{attribute 'GeneratedUsingTerminal: EL2002--0000'}
{attribute addProperty BoxType "EL2002--0000"}
{attribute addProperty Id "WcStateAT %I*BOOL1"}
{attribute addProperty CRC "187373305"}
{attribute addProperty Size "1"}
TYPE WcState_0B2B16F9 :
STRUCT
	{attribute addProperty Name "WcState"}
	WcState AT %I* : BOOL;
END_STRUCT
END_TYPE

(* stored: Version 1.2.0.0, ProductVersion 3.1.4024.11
   DUT WcState_0B2B16F9: Id {8ce21cb7-e99c-4645-b1e7-66eac65636f9} *)
